TYPE EL2869 :
STRUCT
	ch1		:BOOL;
	ch2		:BOOL;
	ch3		:BOOL;
	ch4		:BOOL;
	ch5		:BOOL;
	ch6		:BOOL;
	ch7		:BOOL;
	ch8		:BOOL;
	ch9		:BOOL;
	ch10		:BOOL;
	ch11		:BOOL;
	ch12		:BOOL;
	ch13		:BOOL;
	ch14		:BOOL;
	ch15		:BOOL;
	ch16		:BOOL;	
END_STRUCT
END_TYPE

(* stored: Version 1.1.0.1, ProductVersion 3.1.4024.12
   DUT EL2869: Id {21658651-b5a4-4543-b10e-c027e6e168c1} *)
